Staubli VAL3: WipeCacheRoom2.pgx

program WipeCacheRoom2()
  local num nNum
begin
  for nNum=500 to 999
    sString[nNum]=""
    pfrmCad[nNum].trsf={0,0,0,0,0,0}
  endFor

end
